FUNCTION_BLOCK E_RDELAY (* Reloadable delayed propagation of an event-Cancellable *)
  (* Standard: 61499-1; Classification: Event processing; Description: Copyright (c) 2017 fortiss GmbH This program and the accompanying materials are made available under the terms of the Eclipse Public License 2.0 which is available at https://www.eclipse.org/legal/epl-2.0/ SPDX-License-Identifier: EPL-2.0 *)
  (* Version 1.0, 2017-09-22, Alois Zoitl, fortiss GmbH, initial API and implementation and/or initial documentation *)
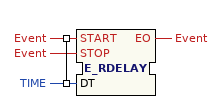
  EVENT_INPUT
    START WITH DT; (* Begin/Reset Delay *)
    STOP; (* Cancel Delay *)
  END_EVENT
  EVENT_OUTPUT
    EO; (* Delayed Event *)
  END_EVENT
  VAR_INPUT
    DT : TIME; (* Delay Time *)
  END_VAR
  SERVICE E_DELAY/RESOURCE (* Reloadable delayed propagation of an event-Cancellable *)
    SEQUENCE event_delay
      E_DELAY.START(DT) -> E_DELAY.EO();
    END_SEQUENCE
    SEQUENCE delay_canceled
      E_DELAY.START(DT);
      E_DELAY.STOP();
    END_SEQUENCE
    SEQUENCE no_multiple_delay
      E_DELAY.START(DT);
      E_DELAY.START(DT);
      -> E_DELAY.EO();
    END_SEQUENCE
  END_SERVICE
END_FUNCTION_BLOCK
